Omron Sysmac Studio project Limit_Kullanimi (Sysmac Studio 1.65.0.64007, StandardProject)

# Controller new_Controller_0: NX1P2-1040DT1 version 1.69
Task PrimaryTask (priority 4, period or condition 2000): Program0

PROGRAM Program0
VAR
    Scale_Valur : ;
    Scale_X0 : Scale_Y0;
    Scale_Y0 : REAL;
    Scale_X1 : REAL;
    Scale_Y1 : REAL;
    Scale_Out : REAL;
    Scale_Value : REAL;
    Lim_Min : REAL;
    Lim_Max : REAL;
    Lim_Out : REAL;
END_VAR

(* Section Section0: ladder, written here as Structured Text *)

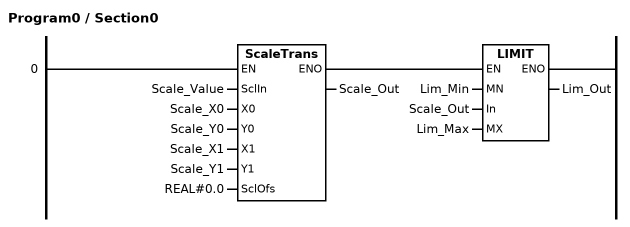
(* Rung 0 *)
Scale_Out := ScaleTrans(SclIn := Scale_Value, X0 := Scale_X0, Y0 := Scale_Y0, X1 := Scale_X1, Y1 := Scale_Y1, SclOfs := REAL#0.0);
Lim_Out := LIMIT(MN := Lim_Min, In := Scale_Out, MX := Lim_Max);
END_PROGRAM